ABB RobotStudio station: Designed_Task.rspag

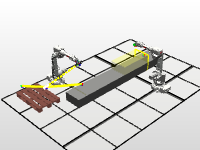
--- station ---
Station Test (saved by RobotStudio 6.8.8148.134)
Controller IRB_2600_12kg_1.65m, task T_ROB1: task frame (RAPID world) sits at (2545.49, 2133.07, 0) mm, rotated rx 0 ry 0 rz 180 deg in the station
Controller System1, task T_ROB1: task frame (RAPID world) sits at (1159.83, 44.08, 0) mm, rotated rx 0 ry 0 rz 90 deg in the station
Controller System1
  mechanical unit ROB_1: IRB2600_12_165_C_01, 6 joints, base frame (-44.08, 1159.83, 0) mm, rotated rx 0 ry 0 rz -90 deg
  mechanical unit CNV1: ?, 1 joints, base frame (-667.31, -410.66, 0) mm
Controller IRB_2600_12kg_1.65m
  mechanical unit ROB_1: IRB2600_12_165_C_01_2, 6 joints, base frame (0, 0, 0) mm
Layout (positions relative to the parent item):
  - SmartComponent_1 [smart component] at (1018.61, 0, 1217.5) mm, rotated rx 180 ry 60 rz 180 deg
      signals: DI Paint, DI Clear
      connections:
        SmartComponent_1.Clear -> PaintApplicator.Clear
        SmartComponent_1.Paint -> PaintApplicator.Enabled
    - PaintApplicator [smart component, from Components\PaintApplicator.rslib] at (0, 0, 69.22) mm, rotated rx 180 ry 0 rz 180 deg
        properties: Part=部件_1; Color=-16777216; ShowPreviewCone=true; Strength=0.1; Range=0.05; Width=0.05; Height=0.05
    - Toolzz [mechanism, from Libraries\Toolzz.rslib] at (0, 0, 0) mm
  - 部件_1 [part] at (1170.48, 576.77, 50) mm
  - IRB2600_12_165_C_01 [mechanism, from Robots\IRB2600_12_165_C_01.rslib] at (0, 0, 0) mm; joint values [0, 0, 0, 0, 0.5236, 0] (rad or m)
  - 输送链 [conveyor] at (1570.48, -2114.95, 0) mm, rotated rx 0 ry 0 rz 90 deg
    - 部件_2 [part] at (691.72, 0, 0) mm
    - 部件_3 [part] at (691.72, 0, 0) mm
    - 传送带对象_6 [conveyorobject] at (1698.51, 0, 0) mm
      - 部件_3 [part]
  - SmartComponent_2 [smart component]
      signals: DO Clear, DO Reached
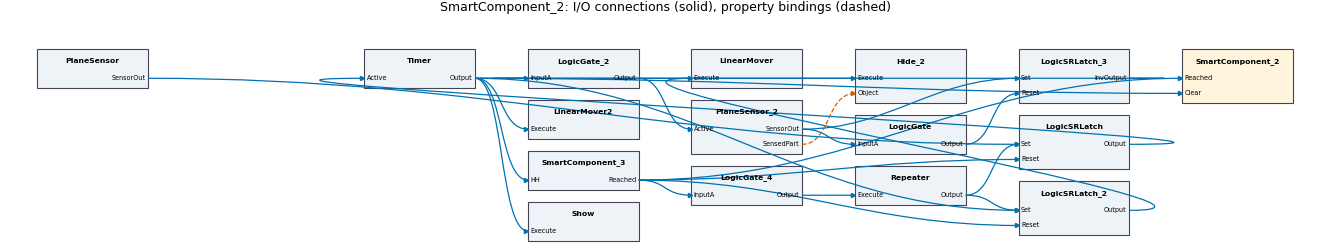
      connections:
        PlaneSensor.SensorOut -> LogicSRLatch.Set
        LogicSRLatch.Output -> Timer.Active
        Timer.Output -> LinearMover2.Execute
        Timer.Output -> LogicSRLatch_2.Set
        PlaneSensor_2.SensorOut -> LogicSRLatch_3.Set
        PlaneSensor_2.SensorOut -> LogicGate.InputA
        LogicGate.Output -> LogicSRLatch_3.Reset
        LogicSRLatch_3.InvOutput -> LogicGate_2.InputA
        LogicGate_2.Output -> PlaneSensor_2.Active
        Timer.Output -> Hide_2.Execute
        Timer.Output -> SmartComponent_3.HH
        SmartComponent_3.Reached -> SmartComponent_2.Reached
        Timer.Output -> SmartComponent_2.Clear
        SmartComponent_3.Reached -> LogicGate_4.InputA
        LogicGate_4.Output -> Repeater.Execute
        SmartComponent_3.Reached -> LogicSRLatch.Reset
        LogicSRLatch_2.Output -> LinearMover.Execute
        SmartComponent_3.Reached -> LogicSRLatch_2.Reset
        Repeater.Output -> LogicSRLatch_2.Set
        Repeater.Output -> LogicSRLatch.Set
        Timer.Output -> Show.Execute
        PlaneSensor_2.SensedPart => Hide_2.Object
    - Timer [smart component, from Components\Timer.rslib]
        properties: StartTime=40; Interval=60; Repeat=true; CurrentTime=0
    - LogicSRLatch [smart component, from Components\LogicSRLatch.rslib]
    - PlaneSensor [smart component, from Components\PlaneSensor.rslib] at (0, -997.88, 0) mm
        properties: Origin=[1.570483 -0.374928018300909 0.32]; Axis1=[-0.6 0 0]; Axis2=[0 0 0.05]; SensedPart=(none)
      - _sensorPart_ [part]
    - LinearMover [smart component, from Components\LinearMover.rslib]
        properties: Object=部件_1; Direction=[0 0.001 0]; Speed=0.02; Reference=Global; ReferenceObject=(none)
    - LogicSRLatch_2 [smart component, from Components\LogicSRLatch.rslib]
    - PlaneSensor_2 [smart component, from Components\PlaneSensor.rslib] at (0, 827.53, 0) mm
        properties: Origin=[1.570483 -1.42322870071312 0.32]; Axis1=[-0.6 0 0]; Axis2=[0 0 0.05]; SensedPart=(none)
      - _sensorPart_ [part]
    - Hide_2 [smart component, from Components\Hide.rslib]
        properties: Object=(none)
    - LogicGate [smart component, from Components\LogicGate.rslib]
        properties: Operator=NOP; Delay=20
    - LogicSRLatch_3 [smart component, from Components\LogicSRLatch.rslib]
    - LogicGate_2 [smart component, from Components\LogicGate.rslib]
        properties: Operator=NOP; Delay=0.1
    - LinearMover2 [smart component, from Components\LinearMover2.rslib]
        properties: Object=部件_1; Direction=[0 -0.001 0]; Distance=1.2; Duration=0; Reference=Global; ReferenceObject=(none)
    - SmartComponent_3 [smart component]
        signals: DI HH, DO Reached
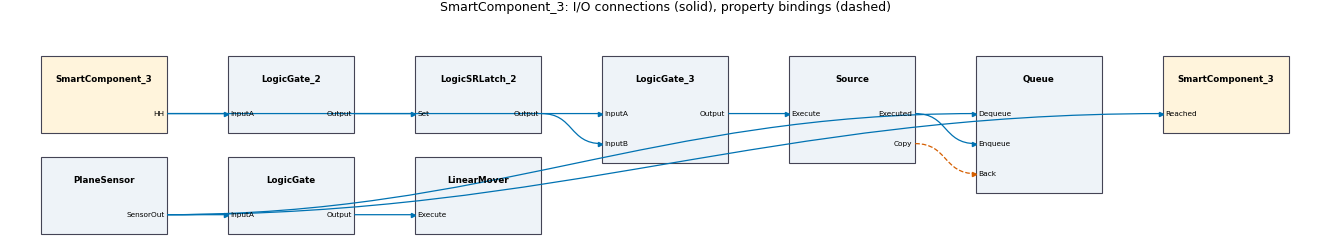
        connections:
          SmartComponent_3.HH -> LogicGate_2.InputA
          LogicGate_2.Output -> LogicSRLatch_2.Set
          SmartComponent_3.HH -> LogicGate_3.InputA
          LogicSRLatch_2.Output -> LogicGate_3.InputB
          LogicGate_3.Output -> Source.Execute
          PlaneSensor.SensorOut -> Queue.Dequeue
          Source.Executed -> Queue.Enqueue
          PlaneSensor.SensorOut -> LogicGate.InputA
          LogicGate.Output -> LinearMover.Execute
          PlaneSensor.SensorOut -> SmartComponent_3.Reached
          Source.Copy => Queue.Back
      - PlaneSensor [smart component, from Components\PlaneSensor.rslib] at (0, 2615.86, 0) mm
          properties: Origin=[1.570483 -0.3358153002911 0.32]; Axis1=[-0.6 0 0]; Axis2=[0 0 0.05]; SensedPart=(none)
        - _sensorPart_ [part]
      - LogicSRLatch_2 [smart component, from Components\LogicSRLatch.rslib]
      - LogicGate [smart component, from Components\LogicGate.rslib]
          properties: Operator=NOT; Delay=0
      - LogicGate_2 [smart component, from Components\LogicGate.rslib]
          properties: Operator=NOP; Delay=0.1
      - LinearMover [smart component, from Components\LinearMover.rslib]
          properties: Object=Queue; Direction=[0 0.001 0]; Speed=0.02; Reference=Global; ReferenceObject=(none)
      - Source [smart component, from Components\Source.rslib]
          properties: Source=部件_2; Copy=(none); Parent=(none); Position=[1.170483 0.576771 0.3]; Orientation=[0 0 0]; Transient=false; PhysicsBehavior=0
      - LogicGate_3 [smart component, from Components\LogicGate.rslib]
          properties: Operator=AND; Delay=0
      - Queue [smart component, from Components\Queue.rslib]
          properties: Back=(none); Front=(none); Queue=; NumberOfObjects=0
    - LogicGate_4 [smart component, from Components\LogicGate.rslib]
        properties: Operator=NOT; Delay=0
    - Repeater [smart component, from Components\Repeater.rslib]
        properties: Count=1
    - Show [smart component, from Components\Show.rslib]
        properties: Object=部件_1
  - 部件_2 [part] at (1880.49, 576.77, 300) mm
  - SmartComponent_4 [smart component]
      connections:
        SimulationEvents.SimulationStarted -> LogicGate.InputA
        LogicGate.Output -> Hide.Execute
        Hide.Executed -> LinearMover2.Execute
    - SimulationEvents [smart component, from Components\SimulationEvents.rslib]
    - LogicGate [smart component, from Components\LogicGate.rslib]
        properties: Operator=NOP; Delay=0.5
    - LinearMover2 [smart component, from Components\LinearMover2.rslib]
        properties: Object=部件_1; Direction=[0 0 0.001]; Distance=0.25; Duration=0; Reference=Global; ReferenceObject=(none)
    - Hide [smart component, from Components\Hide.rslib]
        properties: Object=部件_1
  - IRB2600_12_165_C_01_2 [mechanism, from Robots\IRB2600_12_165_C_01.rslib] at (2545.49, 2133.07, 0) mm, rotated rx 0 ry 0 rz 180 deg; joint values [0, 0, 0, 0, 0.5236, 0] (rad or m)
  - SmartComponent_5 [smart component] at (-290.95, 0, 2016.06) mm, rotated rx 0 ry 60 rz 0 deg
      signals: DI Attach
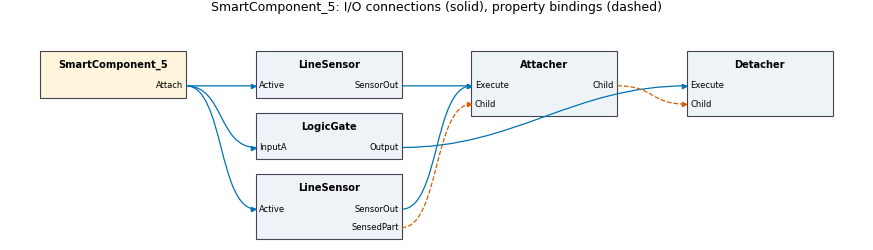
      connections:
        SmartComponent_5.Attach -> LineSensor.Active
        LineSensor.SensorOut -> Attacher.Execute
        SmartComponent_5.Attach -> LogicGate.InputA
        LogicGate.Output -> Detacher.Execute
        SmartComponent_5.Attach -> LineSensor.Active
        LineSensor.SensorOut -> Attacher.Execute
        Attacher.Child => Detacher.Child
        LineSensor.SensedPart => Attacher.Child
    - Xipan [mechanism] at (1601.09, 2132.6, 1175) mm
        TCP Xipan at (0, 0, -95) mm, rotated rx 180 ry 0 rz 180 deg
        links: 吸盘
    - Attacher [smart component, from Components\Attacher.rslib]
        properties: Parent=Xipan; Flange=0; Child=(none); Mount=false; Offset=[0 0 0]; Orientation=[0 0 0]
    - Detacher [smart component, from Components\Detacher.rslib]
        properties: Child=(none); KeepPosition=true
    - LogicGate [smart component, from Components\LogicGate.rslib]
        properties: Operator=NOT; Delay=0
    - LineSensor [smart component, from Components\LineSensor.rslib]
        properties: Start=[1.53109099999999 2.137032 1.04500000000001]; End=[1.53109099999999 2.137032 1.00500000000001]; Radius=0.005; SensedPart=(none); SensedPoint=[0 0 0]
      - _sensorPart_ [part]
  - Euro Pallet [graphiccomponentgroup, from Equipment\Euro Pallet.rslib] at (1615.53, 2766.46, 0) mm
    - Body 1 [part, from Equipment\Euro Pallet.rslib]
Attachment: SmartComponent_1 is attached to IRB2600_12_165_C_01 / Link6
Attachment: SmartComponent_5 is attached to IRB2600_12_165_C_01_2 / Link6
Conveyor tracking 连接: unit CNV1, TravelOffset=0.8, QueueTrackDistance=0, StartWindowWidth=1.2, SyncSeparation=0, CountsPerMeter=10000
Station logic (signal -> signal, property => property):
  SmartComponent_2.Reached -> 输送链.ConveyorStop
  SmartComponent_2.Clear -> SmartComponent_1.Clear
  System1.Paint0 -> SmartComponent_1.Paint
  IRB_2600_12kg_1.65m.do1Attach -> SmartComponent_5.Attach
  SmartComponent_2.Reached -> IRB_2600_12kg_1.65m.di1Reached
Targets, tools, work objects and paths stored in the station and not in the controller backup, written as RAPID:
! task T_ROB1
MODULE Module1
  CONST robtarget Target_30:=[[-44.080184461,78.859448035,1181.499955394],[0.353553391,0.612372436,0.612372436,-0.353553391],[0,0,0,0],[9E+09,9E+09,9E+09,9E+09,9E+09,0]];
ENDMODULE


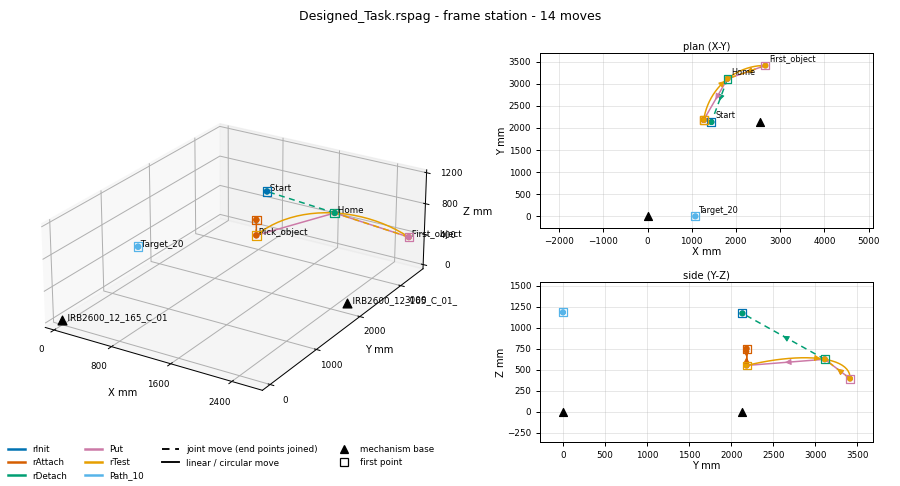
[picture p0: tool path of Designed_Task.rspag in frame station, 14 of 24 moves have a stored position in this frame; points joined in program order, loops and branches not executed]
--- Backups/IRB_2600_12kg_1.65m/RAPID/TASK1/PROGMOD/CalibData.mod ---
MODULE CalibData
	PERS tooldata Xipan:=[TRUE,[[0.603173,0.471776,94.9996],[0,0,0,1]],[1,[0,0,-1],[1,0,0,0],0,0,0]];
ENDMODULE

--- Backups/IRB_2600_12kg_1.65m/RAPID/TASK1/PROGMOD/Module1.mod ---
MODULE Module1
	!CONST robtarget First_object:=[[-120.534304124,-1339.250207991,394.000757409],[-0.000000129,1,0.000000048,0.000000059],[-2,4,-2,0],[9E+09,9E+09,9E+09,9E+09,9E+09,9E+09]];
	!CONST robtarget Pick_object:=[[1275.004967155,-41.385281116,550.375568301],[0.00000001,1,0.000000007,-0.000000001],[-1,0,-1,0],[9E+09,9E+09,9E+09,9E+09,9E+09,9E+09]];
    CONST robtarget Home:=[[737.60463471,-978.55640839,623.895034698],[0.000000013,1,0.000000031,0.000000014],[-1,0,-1,0],[9E+09,9E+09,9E+09,9E+09,9E+09,9E+09]];
    CONST robtarget Middle:=[[630.537946184,-1204.72798405,640.384959144],[0.000000021,1,0.000000156,0.000000057],[-1,0,-1,0],[9E+09,9E+09,9E+09,9E+09,9E+09,9E+09]];
	CONST robtarget Start:=[[1100.58268104,0.47177607,1169.47781335],[0,0.866025404,0,0.5],[0,0,0,0],[9E+09,9E+09,9E+09,9E+09,9E+09,9E+09]];

    VAR robtarget place:=[[0,0,0],[1,0,0,0],[0,0,0,0],[9E+09,9E+09,9E+09,9E+09,9E+09,9E+09]];
    VAR num a:=1;
    CONST robtarget First_object:=[[-120.534131399,-1278.408963951,394.000757409],[0.000000059,1,-0.000000129,0.000000048],[-2,0,-2,0],[9E+09,9E+09,9E+09,9E+09,9E+09,9E+09]];
    CONST robtarget Pick_object:=[[1275.004966194,-48.762460442,550.37559968],[-0.000000008,1,0.000000001,-0.000000009],[-1,0,-1,0],[9E+09,9E+09,9E+09,9E+09,9E+09,9E+09]];

    PROC main()
        rInit;
        WHILE TRUE DO
            WaitDI di1Reached,1;
            rAttach;
            rSetPosition;
            rDetach;
            rSeta;
        ENDWHILE
    ENDPROC

    PROC rInit()
        a:=1;
        Reset do1Attach;
        MoveJ Start,v1000,fine,Xipan\WObj:=wobj0;
    ENDPROC

    PROC rAttach()
        MoveJ offs(Pick_object,0,0,200),v1500,z10,Xipan\WObj:=wobj0;
        MoveL Pick_object,v300,fine,Xipan\WObj:=wobj0;
        set do1Attach;
        WaitTime 1;
        MoveJ offs(Pick_object,0,0,200),v1500,z10,Xipan\WObj:=wobj0;
        !MoveJ Start,v1000,z50,Xipan\WObj:=wobj0;
    ENDPROC

    PROC rDetach()
        !MoveC Home,offs(place,0,0,200),v1000,z100,Xipan\WObj:=wobj0;
        MoveJ offs(place,0,0,200),v1000,z100,Xipan\WObj:=wobj0;
        MoveL place,v300,fine,Xipan\WObj:=wobj0;
        Reset do1Attach;
        WaitTime 1;
        MoveJ offs(place,0,0,200),v1500,z200,Xipan\WObj:=wobj0;
        MoveJ Home,v1000,z100,Xipan\WObj:=wobj0;
        MoveJ Start,v1500,fine,Xipan\WObj:=wobj0;
    ENDPROC

    PROC rSetPosition()
        TEST a
        CASE 1:
        place:=Offs(First_object,0,0,0);
        CASE 2:
        place:=Offs(First_object,200,0,0);
        CASE 3:
        place:=Offs(First_object,400,0,0);
        CASE 4:
        place:=Offs(First_object,600,0,0);
        CASE 5:
        place:=Offs(First_object,0,200,0);
        CASE 6:
        place:=Offs(First_object,200,200,0);
        CASE 7:
        place:=Offs(First_object,400,200,0);
        CASE 8:
        place:=Offs(First_object,600,200,0);
        CASE 9:
        place:=Offs(First_object,0,400,0);
        CASE 10:
        place:=Offs(First_object,200,400,0);
        CASE 11:
        place:=Offs(First_object,400,400,0);
        CASE 12:
        place:=Offs(First_object,600,400,0);
        DEFAULT:
        ENDTEST
    ENDPROC

    PROC rSeta()
        a:=a+1;
        IF a>=13 THEN
            a:=1;
            stop;
        ENDIF
    ENDPROC
    PROC Put()
        MoveL First_object,v1000,z100,Xipan\WObj:=wobj0;
        MoveL Home,v1000,z100,Xipan\WObj:=wobj0;
        MoveL Pick_object,v1000,z100,Xipan\WObj:=wobj0;
    ENDPROC
    PROC rTest()
        MoveJ Pick_object,v1000,z100,Xipan\WObj:=wobj0;
        MoveC Home,First_object,v1000,z100,Xipan\WObj:=wobj0;
        MoveJ Home,v1000,z100,Xipan\WObj:=wobj0;
    ENDPROC

ENDMODULE

--- Backups/System1/RAPID/TASK1/PROGMOD/CalibData.mod ---
MODULE CalibData
	PERS tooldata Toolzz:=[TRUE,[[-5.2839E-5,-6.0885E-5,72.0002],[1,0,0,0]],[1,[0,0,1],[1,0,0,0],0,0,0]];
	TASK PERS wobjdata wobj_cnv1:=[FALSE,FALSE,"CNV1",[[0,0,0],[1,0,0,0]],[[0,0,0],[1,0,0,0]]];
ENDMODULE

--- Backups/System1/RAPID/TASK1/PROGMOD/Module1.mod ---
MODULE Module1
	CONST robtarget Target_20:=[[-44.080184461,78.859448035,1181.499955394],[0.353553391,0.612372436,0.612372436,-0.353553391],[0,0,0,0],[9E+09,9E+09,9E+09,9E+09,9E+09,0]];
	CONST robtarget Target_10:=[[-0.000475335,399.999619367,527.090729268],[0,0.707106781,0.707106781,0],[0,0,0,0],[9E+09,9E+09,9E+09,9E+09,9E+09,0]];

    VAR num x:=0;
    VAR num y:=0;

    PROC main()
        !Add your code here
        ActUnit CNV1;   !??????
        WHILE TRUE DO
            WaitWObj wobj_cnv1; !?????
            Path_10;
            DropWObj wobj_cnv1; !??????

        ENDWHILE
    ENDPROC

	PROC Path_10()
        MoveL Target_20,v800,z100,Toolzz\WObj:=wobj0;
        x:=0;
        MoveL Offs(Target_10,0,x,0),v800,fine,Toolzz\WObj:=wobj_cnv1;
        SetDO Paint0,1;
        FOR i FROM 1 TO 5 DO
            MoveL Offs(Target_10,0,x,0),v80,fine,Toolzz\WObj:=wobj_cnv1;
            MoveL Offs(Target_10,200,x,0),v80,fine,Toolzz\WObj:=wobj_cnv1;
            x:=x-20;
            MoveL Offs(Target_10,200,x,0),v80,fine,Toolzz\WObj:=wobj_cnv1;
            MoveL Offs(Target_10,0,x,0),v80,fine,Toolzz\WObj:=wobj_cnv1;
            x:=x-20;

        ENDFOR

        MoveL Offs(Target_10,0,x,0),v80,fine,Toolzz\WObj:=wobj_cnv1;
        MoveL Offs(Target_10,200,x,0),v80,fine,Toolzz\WObj:=wobj_cnv1;


        SetDO Paint0,0;
	    MoveL Target_20,v800,z100,Toolzz\WObj:=wobj0;
	    !MoveL Target_10,v1000,z100,Toolzz\WObj:=wobj_cnv1;
	ENDPROC
ENDMODULE

--- Backups/IRB_2600_12kg_1.65m/SYSPAR/EIO.cfg ---
EIO:CFG_1.0:6:1::
#
INDUSTRIAL_NETWORK:

      -Name "DeviceNet" -Label "DeviceNet Master/Slave Network" -Address "2"
#
DEVICENET_DEVICE:

      -Name "d652" -VendorName "ABB Robotics" -ProductName "24 VDC I/O Device"\
      -Label "DSQC 652 24 VDC I/O Device" -Address 10 -ProductCode 26\
      -DeviceType 7 -ConnectionType "COS" -OutputSize 2 -InputSize 2
#
DEVICENET_INTERNAL_DEVICE:

      -Name "DN_Internal_Device" -VendorName "ABB Robotics"\
      -ProductName "DeviceNet Internal Slave Device"
#
EIO_SIGNAL:

      -Name "do1Attach" -SignalType "DO" -Device "d652" -DeviceMap "0"

      -Name "di1Reached" -SignalType "DI" -Device "d652" -DeviceMap "0"

--- Backups/System1/SYSPAR/EIO.cfg ---
EIO:CFG_1.0:6:1::
#
INDUSTRIAL_NETWORK:

      -Name "RobICI" -Label "RobICI Network"
#
ROBICI_DEVICE:

      -Name "CTM1" -TrustLevel "InternalDeviceTrustLevel"\
      -VendorName "ABB Robotics" -ProductName "DSQC2000"\
      -Label "Conveyor Tracking Device 1" -Address "0.0.0.0"
#
EIO_SIGNAL:

      -Name "c1Counts" -SignalType "GI" -Device "CTM1"\
      -DeviceMap "Enc1:position"

      -Name "c1CountsPerSec" -SignalType "AI" -Device "CTM1"\
      -DeviceMap "Enc1:velocity"

      -Name "c1TrigVis" -SignalType "DO" -Device "CTM1" -Label "Trig X21 pin 5"\
      -DeviceMap "Digout1:Setpoint"

      -Name "c1TrigAutoMode" -SignalType "DO" -Device "CTM1"\
      -DeviceMap "Cam1:Connect"

      -Name "c1TrigAutoDist" -SignalType "GO" -Device "CTM1"\
      -DeviceMap "Cam1:Interval"

      -Name "c1TrigAutoEncNo" -SignalType "GO" -Device "CTM1"\
      -DeviceMap "Cam1Enc:DeviceNo"

      -Name "c1CntFromEnc" -SignalType "GI" -Device "CTM1"\
      -DeviceMap "Sync1Enc1:Value"

      -Name "c1SoftSync" -SignalType "DO" -Device "CTM1"\
      -DeviceMap "Sync1Enc1:SyncTrig"

      -Name "c1SpeedBandWidth" -SignalType "GI" -Device "CTM1"\
      -DeviceMap "e1_SpeedBandWidth:SetPoint"

      -Name "c1Position" -SignalType "AO" -MaxLog 21474.8 -MaxPhys 1\
      -MaxPhysLimit 1 -MaxBitVal 2147483647 -MinLog -21474.8 -MinPhys -1\
      -MinPhysLimit -1 -MinBitVal -2147483647 -Size 32

      -Name "c1Speed" -SignalType "AO" -MaxLog 21474.8 -MaxPhys 1\
      -MaxPhysLimit 1 -MaxBitVal 2147483647 -MinLog -21474.8 -MinPhys -1\
      -MinPhysLimit -1 -MinBitVal -2147483647 -Size 32

      -Name "c1Connected" -SignalType "DO"

      -Name "c1NullSpeed" -SignalType "DO"

      -Name "c1PassStw" -SignalType "DO"

      -Name "c1NewObjStrobe" -SignalType "DO"

      -Name "c1WaitWObj" -SignalType "DO"

      -Name "c1DropWObj" -SignalType "DO" -Access "ALL"

      -Name "c1Rem1PObj" -SignalType "DO" -Access "All"

      -Name "c1RemAllPObj" -SignalType "DO" -Access "All"

      -Name "c1CntToEncStr" -SignalType "DO"

      -Name "c1PosInJobQ" -SignalType "DO" -Default 1

      -Name "c1ObjectsInQ" -SignalType "GO" -Size 8

      -Name "c1CntToEnc" -SignalType "GO" -Size 32

      -Name "Paint0" -SignalType "DO"

--- Backups/System1/SYSPAR/PROC.cfg ---
PROC:CFG_1.0:6:0::
#
CONVEYOR:

      -name "CNV1" -sensor_type "ICI" -use_sensor "ICI1" -adjustment_speed 850\
      -min_dist -600 -max_dist 20000 -correction_vector_ramp_length 5
#
CONVEYOR_ICI_SENSOR:

      -name "ICI1" -connected_signal "c1Connected" -position_signal "c1Position"\
      -velocity_signal "c1Speed" -position_count_signal "c1Counts"\
      -velocity_count_signal "c1CountsPerSec" -null_speed_signal "c1NullSpeed"\
      -wait_wobj_signal "c1WaitWObj" -drop_wobj_signal "c1DropWObj"\
      -rem_all_pobj_signal "c1RemAllPObj" -rem_one_pobj_signal "c1Rem1PObj"\
      -supervise_max_dist_off  -newobj_strobe "c1NewObjStrobe"\
      -count_to_enc_strobe "c1CntToEncStr" -obj_in_queue_signal "c1ObjectsInQ"\
      -count_from_enc "c1CntFromEnc" -count_to_enc "c1CntToEnc"\
      -StartWinWidth 1.2 -speed_filter_bandwidth "c1SpeedBandWidth"
